Staubli VAL3: remErrManual.pgx

program remErrManual(string& sReturn[] (dimensions=1))
begin
  // Error raised when we attempt a remote-only command in manual mode
  //
  logMsg("call remErrManual")
  sReturn="ERROR 402"
  sReturn=sReturn+": Abort cmd, not in remote mode."
  logMsg(sReturn)
end
